FUNCTION_BLOCK FB_eventRingBuffer
VAR
	bufferRingArray : ARRAY[1..20] OF ST_Event;
	headIndex : INT := 1;
	tailIndex : INT := 1;
	currentPosition : INT := 1;
	
END_VAR
VAR CONSTANT
	ringBufferSize : INT := 20;
END_VAR

METHOD Apend : BOOL
VAR_INPUT
	stEvent : ST_Event;
END_VAR
IF currentPosition >= ringBufferSize THEN
	Apend:= FALSE;
ELSE
	bufferRingArray[headIndex]:= stEvent;		
	headIndex := headIndex+1;
	currentPosition:=currentPosition+1;
	Apend:= True;
END_IF
END_METHOD

METHOD Remove : BOOL
VAR_OUTPUT
	stEvent: ST_Event;
END_VAR
IF currentPosition:=0 THEN
	Remove:= FALSE;
ELSE
	stEvent:= bufferRingArray[currentPosition];
	tailIndex:= tailIndex+1;
	currentPosition:= currentPosition-1;
	Remove:= TRUE;
END_IF
END_METHOD

END_FUNCTION_BLOCK

(* stored: Version 1.1.0.1, ProductVersion 3.1.4024.16
   POU FB_EventRingBuffer: Id {79d13302-3958-48fe-96d8-2afbac72a2d0}, SpecialFunc None
   Method Apend: Id {5b1cde54-9656-42c6-9317-400f7ce8851a}
   Method Remove: Id {013e1d0a-326c-4d96-b493-210e65f797d3} *)
